Yaskawa INFORM job: AAA.JBI

/JOB
//NAME AAA
//POS
///NPOS 3,0,0,0,0,0
C00000=-49439,115900,74994,3819,-53506,-4422
C00001=-47805,108597,65281,4512,-51369,-5178
C00002=-46969,105372,61036,4871,-50464,-5567
//INST
///DATE 2023/01/24 13:34
///ATTR SC,RW
///GROUP1 RB1
NOP
MOVL C00000 V=10.0 PL=8
ARCON
MOVL C00001 V=10.0 PL=8
ARCOF
MOVL C00002 V=10.0 PL=8
END
